Yaskawa INFORM job: OK_R2_O34-37(210,0_180)2AWOK.JBI

/JOB
//NAME OK_R2_O34-37(210,0_180)2AWOK
///FOLDERNAME X4
//POS
///NPOS 226,226,226,7,0,0
///TOOL 0
///POSTYPE PULSE
///PULSE
C00000=-125700,-80476,-34247,159249,27287,28453
C00001=-123130,-74105,-30702,162391,25597,27223
C00002=-122202,-71536,-29217,163608,24992,26738
C00003=-121293,-68396,-25015,165796,25706,25775
C00004=-119897,-67278,-25144,167731,24799,24999
C00005=-121293,-68396,-25015,165796,25706,25775
C00006=-122202,-71536,-29217,163608,24992,26738
C00007=-123284,-67899,-27862,160952,24298,27913
C00008=-122447,-67212,-26586,162727,24486,27140
C00009=-123284,-67899,-27862,160952,24298,27913
C00010=-122202,-71536,-29217,163608,24992,26738
C00011=-123130,-74105,-30702,162391,25597,27223
C00012=-125700,-80476,-34247,159249,27287,28453
C00013=-125517,-80437,-34211,159525,27238,28339
C00014=-122961,-74061,-30663,162666,25556,27108
C00015=-122038,-71489,-29176,163883,24954,26623
C00016=-117667,-71002,-28856,171434,24065,23454
C00017=-117704,-70431,-28835,171227,23800,23550
C00018=-117667,-71002,-28856,171434,24065,23454
C00019=-122038,-71489,-29176,163883,24954,26623
C00020=-119799,-70680,-31927,166276,22459,25716
C00021=-118976,-69928,-30572,168119,22724,24911
C00022=-119799,-70680,-31927,166276,22459,25716
C00023=-122038,-71489,-29176,163883,24954,26623
C00024=-122961,-74061,-30663,162666,25556,27108
C00025=-125517,-80437,-34211,159525,27238,28339
C00026=-140387,-129911,-44763,153839,48320,28262
C00027=-154667,-139794,-63765,132481,63225,34326
C00028=-155865,-52236,-95522,47063,99015,61474
C00029=-122410,-67393,-33433,34982,73766,64939
C00030=-118917,-73983,-33918,35626,69830,65070
C00031=-118508,-70070,-27252,36089,67956,64591
C00032=-117264,-69435,-26201,36204,67200,64847
C00033=-118508,-70070,-27252,36089,67956,64591
C00034=-118437,-72039,-27377,36310,67165,64343
C00035=-118508,-70070,-27252,36089,67956,64591
C00036=-123060,-73487,-31863,35667,70648,63634
C00037=-125159,-74654,-36532,35162,73351,63677
C00038=-117818,-78878,-43515,44751,78217,64927
C00039=-114758,-78477,-39683,45348,75169,64953
C00040=-113298,-77876,-37428,45678,73684,64940
C00041=-114862,-79533,-39394,45465,74705,64688
C00042=-113645,-77017,-38294,45463,74548,65185
C00043=-113477,-77789,-37161,45383,73476,65293
C00044=-119505,-70896,-29485,43711,74626,65290
C00045=-120144,-69706,-28375,43648,74873,65114
C00046=-125052,-63057,-20955,43194,76309,63552
C00047=-128321,-58110,-15632,44166,78560,60322
C00048=-131102,-53426,-10460,43738,79284,59417
C00049=-129277,-58077,-17153,43886,79704,60402
C00050=-131618,-58273,-21031,43272,82484,60567
C00051=-155865,-52236,-95522,47063,99015,61474
C00052=-107841,-78990,-100274,15174,85565,25314
C00053=-120644,-33075,-33747,-17198,86743,-72858
C00054=-120645,-33066,-33740,-17198,86743,-72858
C00055=-121261,-33537,-33634,-17157,86319,-73016
C00056=-120651,-31294,-33185,-17194,87287,-72936
C00057=-120265,-34286,-35568,-17221,87300,-72802
C00058=-121246,-33499,-33406,-17160,86207,-72996
C00059=-120695,-32982,-32791,-17199,86212,-72803
C00060=-123405,-31941,-32460,-10145,86277,-73561
C00061=-120644,-33063,-33738,-17198,86744,-72858
C00062=-120644,-33063,-33738,-17198,86744,-72858
C00063=-120644,-33085,-33753,-9248,85868,-74516
C00064=-120658,-33883,-52020,3249,107968,-57945
C00065=-120634,-51653,-31257,6589,89487,-53974
C00066=-120887,-59194,-41100,6571,91677,-53945
C00067=-114365,-59297,-40540,7297,90721,-51781
C00068=-121686,-52648,-32529,6467,89842,-54312
C00069=-120641,-50150,-31062,6590,90137,-53943
C00070=-115090,-58916,-39821,7220,90542,-52038
C00071=-121020,-51343,-30297,6544,89092,-54127
C00072=-121570,-70600,-40611,7004,74168,-55148
C00073=-127404,-59840,-28957,5949,73181,-57087
C00074=-128623,-57920,-26766,5993,72907,-57518
C00075=-120636,-51546,-31197,-12806,84757,-45971
C00076=-120635,-51562,-31206,-12806,84754,-45970
C00077=-120637,-51473,-31156,-31547,98354,-39015
C00078=-120638,-51464,-31151,-31547,98355,-39016
C00079=-127651,-66621,-42293,-29165,87585,-39205
C00080=-120645,-49986,-30969,-31614,98908,-39175
C00081=-120184,-52981,-33063,-31488,98864,-38978
C00082=-126387,-66657,-42132,-29030,87918,-38805
C00083=-124162,-65853,-41061,-28777,88461,-38095
C00084=-123779,-65431,-40746,-28731,88612,-37988
C00085=-116886,-63013,-38039,-27795,90542,-35857
C00086=-116876,-68393,-50736,-27992,95034,-36929
C00087=-127335,-91521,-66356,2133,76505,-53999
C00088=-120632,-51605,-31230,12938,89151,-58072
C00089=-122382,-77541,-49676,15704,77889,-41459
C00090=-116417,-82504,-50333,15734,74684,-39769
C00091=-121684,-52600,-32501,12821,89583,-58390
C00092=-120640,-50101,-31034,12940,89789,-58008
C00093=-117566,-82113,-49782,15768,74770,-40162
C00094=-137736,-66681,-32025,26351,79133,-47852
C00095=-137780,-65826,-31188,26317,79067,-47879
C00096=-127334,-50999,-24101,13599,84251,-46609
C00097=-127274,-55905,-35607,13545,88687,-46195
C00098=-120633,-51614,-31235,12938,89150,-58073
C00099=-120634,-51391,-31110,-31547,98367,-39018
C00100=-120635,-51381,-31104,-31548,98368,-39018
C00101=-123679,-52106,-31631,-32185,97183,-39896
C00102=-120642,-49903,-30922,-31614,98921,-39177
C00103=-120181,-52898,-33017,-31489,98878,-38981
C00104=-120835,-59376,-36016,-31166,93226,-37672
C00105=-121613,-72530,-44193,-30286,84455,-35757
C00106=-118747,-61104,-37303,-26246,91458,-36794
C00107=-120635,-51379,-31103,-26471,93957,-42710
C00108=-120633,-51391,-31110,-26470,93955,-42709
C00109=-120630,-51586,-31219,10910,92232,-53915
C00110=-120632,-51644,-31252,6564,89533,-53910
C00111=-103812,-53067,-78891,-39071,105659,-38988
C00112=-91163,-136711,-112609,-36408,93269,-29237
C00113=-91163,-136711,-112609,-36408,93269,-29237
C00114=-91163,-136711,-112609,-36408,93269,-29237
C00115=-91163,-136711,-112609,-36408,93269,-29237
C00116=-14735,-147183,-53705,-96059,99176,-32960
C00117=-116063,-75069,-24786,-161373,30180,-27192
C00118=-118646,-74586,-30917,-162370,25797,-27057
C00119=-119577,-72016,-29437,-163583,25187,-26574
C00120=-122851,-69134,-26289,-169408,24955,-24114
C00121=-122803,-67500,-26251,-168862,24172,-24377
C00122=-122851,-69134,-26289,-169408,24955,-24114
C00123=-119577,-72016,-29437,-163583,25187,-26574
C00124=-119782,-71043,-35943,-152224,16280,-31420
C00125=-121147,-70052,-34044,-156561,16387,-29537
C00126=-119067,-67658,-29205,-160988,23362,-27785
C00127=-119577,-72016,-29437,-163583,25187,-26574
C00128=-118646,-74586,-30917,-162370,25797,-27057
C00129=-116063,-80958,-34447,-159238,27499,-28281
C00130=-116167,-79884,-33984,-159178,27227,-28326
C00131=-118709,-73507,-30415,-162283,25553,-27108
C00132=-119627,-70935,-28920,-163488,24953,-26627
C00133=-124970,-68554,-27226,-172714,23781,-22752
C00134=-124929,-67933,-27226,-172492,23472,-22855
C00135=-124970,-68554,-27226,-172714,23781,-22752
C00136=-119627,-70935,-28920,-163488,24953,-26627
C00137=-114841,-73408,-48022,-82057,16864,-69970
C00138=-115635,-73012,-47011,-83260,16231,-69454
C00139=-119724,-68827,-29398,-162557,23640,-27094
C00140=-119627,-70935,-28920,-163488,24953,-26627
C00141=-118709,-73507,-30415,-162283,25553,-27108
C00142=-116167,-79884,-33984,-159178,27227,-28326
C00143=-99237,-131925,-44709,-152289,49940,-28409
C00144=-62709,-186403,-96766,-116405,74373,-39052
C00145=-70314,-132957,-105748,-65746,79738,-62154
C00146=-61806,-120643,-118554,-32165,89559,-74963
C00147=-100254,-58589,-20850,-47462,84028,-58675
C00148=-101968,-51866,-3168,-48574,78104,-56512
C00149=-101968,-51553,-2632,-48598,77990,-56453
C00150=-101518,-52976,-2809,-48578,77787,-56140
C00151=-101968,-51553,-2632,-48598,77990,-56453
C00152=-103386,-50149,-432,-49034,76876,-56530
C00153=-101968,-51553,-2632,-48598,77990,-56453
C00154=-100254,-58589,-20850,-47462,84028,-58675
C00155=-120623,-69117,-28104,-48531,104993,-26022
C00156=-124022,-87503,-41913,-47197,93373,-21899
C00157=-120632,-67990,-28310,-48704,105465,-26277
C00158=-119274,-70289,-29410,-48044,105816,-25785
C00159=-123549,-87206,-41537,-47050,93555,-21770
C00160=-115351,-77678,-31893,-44276,96770,-19561
C00161=-115180,-76774,-30982,-44204,96783,-19491
C00162=-107611,-66250,-20317,-41245,99360,-17323
C00163=-104022,-60066,-14079,-39703,100393,-16240
C00164=-107611,-77742,-40705,-42371,104385,-19399
C00165=-61806,-120643,-118554,-32165,89559,-74963
C00166=-96268,-101177,-113144,-8865,97124,-11070
C00167=-120641,-42853,-51550,17560,92173,73840
C00168=-120646,-33870,-34272,17525,86425,73017
C00169=-119942,-58321,-47290,17224,67969,70679
C00170=-121031,-35101,-36097,17549,86977,72960
C00171=-120651,-32098,-33726,17520,86975,73094
C00172=-121087,-58091,-46777,17546,68025,70253
C00173=-122899,-57278,-45773,18035,68227,69595
C00174=-123358,-56945,-45288,18164,68208,69418
C00175=-121878,-55895,-44787,12232,67936,69995
C00176=-118961,-54720,-57543,10936,75808,71809
C00177=-120654,-86347,-59671,-2864,63718,59361
C00178=-125912,-56068,-36753,-6250,87624,52842
C00179=-128066,-58011,-42816,-6649,92655,51740
C00180=-129226,-58813,-41203,-6752,91180,51406
C00181=-120642,-50370,-31189,-6165,90024,54116
C00182=-119584,-52858,-32650,-6041,89726,54489
C00183=-128796,-58655,-40767,-6707,91029,51560
C00184=-122766,-51369,-31065,-6034,89291,53691
C00185=-122762,-63238,-38041,-5894,80464,54098
C00186=-119550,-58975,-32943,-5845,79752,55225
C00187=-122768,-60053,-29242,1998,72011,53401
C00188=-124703,-66651,-43936,2040,77707,52830
C00189=-120638,-51944,-31419,32003,97998,39113
C00190=-120639,-51928,-31410,32003,98001,39113
C00191=-118996,-52516,-31682,32334,97265,39558
C00192=-121098,-53452,-33319,31944,98508,39075
C00193=-120645,-50452,-31236,32066,98559,39271
C00194=-119173,-52749,-31833,32295,97308,39501
C00195=-119801,-52482,-32070,32192,97780,39386
C00196=-119899,-52107,-31634,32164,97752,39338
C00197=-119950,-60824,-38736,26131,92333,38222
C00198=-119950,-65442,-50997,26401,96995,39269
C00199=-116899,-68263,-56336,11454,97179,48279
C00200=-127404,-81706,-52066,-14147,73081,57801
C00201=-116720,-79858,-46664,-24697,73771,62487
C00202=-120640,-50459,-31240,-12516,89696,58190
C00203=-119581,-52948,-32700,-12396,89486,58575
C00204=-115512,-79082,-45759,-25163,74038,62927
C00205=-108001,-68814,-34854,-26331,75228,65611
C00206=-108064,-68383,-34491,-26332,75206,65593
C00207=-103624,-60475,-25996,-26279,75513,67180
C00208=-112718,-64474,-31424,-18064,72408,63442
C00209=-112718,-70905,-44852,-17685,77140,62731
C00210=-112718,-71186,-45475,-17671,77368,62698
C00211=-120385,-74764,-48938,3443,103646,-6733
C00212=-120303,-75998,-49738,3392,102861,-6716
C00213=-118985,-76178,-48936,3795,102220,-6275
C00214=-121095,-53483,-33336,3688,117233,-6601
C00215=-120643,-50483,-31254,3935,117471,-6417
C00216=-122593,-74979,-47472,2658,102081,-7526
C00217=-122814,-74696,-47089,2584,101998,-7604
C00218=-129478,-71737,-44300,477,101932,-9900
C00219=-129478,-75128,-51887,483,104859,-9888
C00220=-120632,-52031,-31468,10348,93078,-4644
C00221=-120631,-51970,-31434,-12514,89052,58257
C00222=-126964,-95845,-81485,3515,87950,51222
C00223=-130419,-125155,-112371,3575,92040,50165
C00224=-16344,-125828,-114775,3579,93173,50196
C00225=-16344,-125828,-114775,3579,93173,50196
BC00000=299799,668083,634815
BC00001=299799,668083,634815
BC00002=299799,668083,634815
BC00003=299799,668083,634815
BC00004=299799,668083,634815
BC00005=299799,668083,634815
BC00006=299799,668083,634815
BC00007=299799,668083,634815
BC00008=299799,668083,634815
BC00009=299799,668083,634815
BC00010=299799,668083,634815
BC00011=299799,668083,634815
BC00012=299799,668083,634815
BC00013=258861,679019,566863
BC00014=258861,679019,566863
BC00015=258861,679019,566863
BC00016=258861,679019,566863
BC00017=258861,679019,566863
BC00018=258861,679019,566863
BC00019=258861,679019,566863
BC00020=258861,679019,566863
BC00021=258861,679019,566863
BC00022=258861,679019,566863
BC00023=258861,679019,566863
BC00024=258861,679019,566863
BC00025=258861,679019,566863
BC00026=258861,679019,566863
BC00027=246190,684484,603571
BC00028=168329,718064,829131
BC00029=168329,806325,829131
BC00030=168329,806325,829131
BC00031=168329,806325,829131
BC00032=168329,806325,829131
BC00033=168329,806325,829131
BC00034=168329,806325,829131
BC00035=168329,806325,829131
BC00036=168329,806325,829131
BC00037=168329,806325,829131
BC00038=161625,808865,790208
BC00039=161625,808865,790208
BC00040=161625,808865,790208
BC00041=161625,808865,790208
BC00042=161625,808865,790208
BC00043=161625,808865,790208
BC00044=161625,808865,790208
BC00045=161625,808865,790208
BC00046=161625,808865,790208
BC00047=161625,808865,790208
BC00048=161625,808865,790208
BC00049=161625,808865,790208
BC00050=161625,808865,790208
BC00051=168329,718064,829131
BC00052=233669,718722,855431
BC00053=356753,719962,904973
BC00054=355561,717940,879352
BC00055=355084,717131,869103
BC00056=355084,717131,869103
BC00057=355084,717131,869103
BC00058=358688,717759,865405
BC00059=358688,717759,865405
BC00060=358688,717759,865405
BC00061=360357,720590,901274
BC00062=360145,720879,899518
BC00063=353052,720476,901588
BC00064=275657,749180,834890
BC00065=252725,782753,902871
BC00066=256148,780353,880096
BC00067=257517,779394,870985
BC00068=257517,779394,870985
BC00069=257517,779394,870985
BC00070=257517,779394,870985
BC00071=257517,779394,870985
BC00072=257517,779394,870985
BC00073=257517,779394,870985
BC00074=257517,779394,870985
BC00075=279626,776550,839590
BC00076=278375,777634,865867
BC00077=302522,799758,822544
BC00078=301330,797736,796923
BC00079=300854,796928,786673
BC00080=300853,796927,786675
BC00081=300853,796927,786675
BC00082=300854,796928,786673
BC00083=300854,796928,786673
BC00084=300854,796928,786673
BC00085=300854,796928,786673
BC00086=300854,796928,786673
BC00087=285946,783794,900084
BC00088=276545,775017,942522
BC00089=280455,772329,921075
BC00090=280455,772329,921075
BC00091=282019,771253,912497
BC00092=282019,771253,912497
BC00093=280455,772329,921075
BC00094=280455,772329,921075
BC00095=280455,772329,921075
BC00096=280455,772329,921075
BC00097=280403,772359,920891
BC00098=268658,779616,914487
BC00099=344074,788201,893588
BC00100=342882,786179,867967
BC00101=342405,785370,857718
BC00102=342405,785370,857718
BC00103=342405,785370,857718
BC00104=342405,785370,857718
BC00105=342405,785370,857718
BC00106=342405,785370,857718
BC00107=345131,781299,876890
BC00108=345652,783183,902892
BC00109=289564,773957,978220
BC00110=261789,777074,937860
BC00111=353536,737917,894599
BC00112=353536,695664,894599
BC00113=353536,695664,894599
BC00114=353536,695664,894599
BC00115=353536,695664,894599
BC00116=166023,670483,663813
BC00117=139859,666970,631611
BC00118=139859,666970,631611
BC00119=139859,666970,631611
BC00120=139859,666970,631611
BC00121=139859,666971,631609
BC00122=139859,666970,631611
BC00123=139859,666970,631611
BC00124=139859,666970,631611
BC00125=139859,666970,631609
BC00126=139859,666970,631611
BC00127=139859,666970,631611
BC00128=139859,666970,631611
BC00129=139859,666970,631611
BC00130=178204,675740,573402
BC00131=178204,675740,573402
BC00132=178204,675740,573402
BC00133=178204,675740,573402
BC00134=178204,675740,573402
BC00135=178204,675740,573402
BC00136=178204,675740,573402
BC00137=178204,675740,573402
BC00138=178204,675740,573402
BC00139=178204,675740,573402
BC00140=178204,675740,573402
BC00141=178204,675740,573402
BC00142=178204,675740,573402
BC00143=178204,675740,573402
BC00144=191883,696660,621052
BC00145=236191,764425,852086
BC00146=260221,801176,958847
BC00147=260221,801176,859111
BC00148=260221,801176,859108
BC00149=260221,801176,859108
BC00150=260221,801176,859108
BC00151=260221,801176,859108
BC00152=260221,801176,859108
BC00153=260221,801176,859108
BC00154=260221,801176,859111
BC00155=271447,845610,763612
BC00156=269989,844590,755462
BC00157=269905,844531,754994
BC00158=269905,844531,754994
BC00159=269989,844590,755462
BC00160=269989,844590,755462
BC00161=269989,844590,755462
BC00162=269989,844590,755462
BC00163=269989,844590,755462
BC00164=269989,844590,755462
BC00165=260221,801176,859111
BC00166=179215,763567,877996
BC00167=81732,718309,900722
BC00168=82982,716309,875111
BC00169=83482,715509,864866
BC00170=83482,715509,864866
BC00171=83482,715509,864866
BC00172=83482,715509,864866
BC00173=83482,715509,864866
BC00174=83482,715509,864866
BC00175=83482,715509,864866
BC00176=83482,715509,864866
BC00177=162723,767201,899794
BC00178=183133,779963,900503
BC00179=180774,777935,868378
BC00180=180772,777936,868380
BC00181=180651,777993,868574
BC00182=180651,777993,868574
BC00183=180772,777936,868380
BC00184=180772,777936,868380
BC00185=180772,777936,868380
BC00186=180772,777936,868380
BC00187=180772,777936,868380
BC00188=180772,777936,868380
BC00189=135124,798065,819777
BC00190=136374,796066,794166
BC00191=136671,795591,788088
BC00192=136874,795266,783921
BC00193=136874,795266,783921
BC00194=136199,795636,787117
BC00195=132017,796135,779854
BC00196=132017,796135,779854
BC00197=132017,796135,779854
BC00198=132017,796135,779854
BC00199=143790,787140,843333
BC00200=157760,770823,917898
BC00201=157760,770823,917898
BC00202=156218,769744,909280
BC00203=156218,769744,909280
BC00204=157760,770823,917898
BC00205=157760,770824,917897
BC00206=157760,770824,917897
BC00207=157760,770824,917897
BC00208=157760,770824,917897
BC00209=157760,770824,917897
BC00210=157760,770824,917897
BC00211=135405,814938,885725
BC00212=136655,812939,860113
BC00213=136655,812939,860113
BC00214=137155,812139,849869
BC00215=137155,812139,849869
BC00216=136655,812939,860113
BC00217=136655,812939,860113
BC00218=136655,812939,860113
BC00219=136655,812939,860113
BC00220=125409,766237,942300
BC00221=152567,767692,974231
BC00222=182902,779158,882705
BC00223=182902,779158,882705
BC00224=182902,779158,882705
BC00225=182902,668970,882705
EC00000=1862365,0
EC00001=1862365,0
EC00002=1862365,0
EC00003=1862365,0
EC00004=1862365,0
EC00005=1862365,0
EC00006=1862365,0
EC00007=1862365,0
EC00008=1862365,0
EC00009=1862365,0
EC00010=1862365,0
EC00011=1862365,0
EC00012=1862365,0
EC00013=1862365,0
EC00014=1862365,0
EC00015=1862365,0
EC00016=1862365,0
EC00017=1862365,0
EC00018=1862365,0
EC00019=1862365,0
EC00020=1862365,0
EC00021=1862365,0
EC00022=1862365,0
EC00023=1862365,0
EC00024=1862365,0
EC00025=1862365,0
EC00026=1862365,0
EC00027=1862365,0
EC00028=1862365,0
EC00029=1862365,0
EC00030=1862365,0
EC00031=1862365,0
EC00032=1862365,0
EC00033=1862365,0
EC00034=1862365,0
EC00035=1862365,0
EC00036=1862365,0
EC00037=1862365,0
EC00038=1862365,0
EC00039=1862365,0
EC00040=1862365,0
EC00041=1862365,0
EC00042=1862365,0
EC00043=1862365,0
EC00044=1862365,0
EC00045=1862365,0
EC00046=1862365,0
EC00047=1862365,0
EC00048=1862365,0
EC00049=1862365,0
EC00050=1862365,0
EC00051=1862365,0
EC00052=1862365,0
EC00053=1862365,0
EC00054=1862365,0
EC00055=1862365,0
EC00056=1862365,0
EC00057=1862365,0
EC00058=1862365,0
EC00059=1862365,0
EC00060=1862365,0
EC00061=1862365,0
EC00062=1862365,0
EC00063=1862365,0
EC00064=1862365,0
EC00065=1862365,0
EC00066=1862365,0
EC00067=1862365,0
EC00068=1862365,0
EC00069=1862365,0
EC00070=1862365,0
EC00071=1862365,0
EC00072=1862365,0
EC00073=1862365,0
EC00074=1862365,0
EC00075=1862365,0
EC00076=1862365,0
EC00077=1862365,0
EC00078=1862365,0
EC00079=1862365,0
EC00080=1862365,0
EC00081=1862365,0
EC00082=1862365,0
EC00083=1862365,0
EC00084=1862365,0
EC00085=1862365,0
EC00086=1862365,0
EC00087=1862365,0
EC00088=1862365,0
EC00089=1862365,0
EC00090=1862365,0
EC00091=1862365,0
EC00092=1862365,0
EC00093=1862365,0
EC00094=1862365,0
EC00095=1862365,0
EC00096=1862365,0
EC00097=1862365,0
EC00098=1862365,0
EC00099=1862365,0
EC00100=1862365,0
EC00101=1862365,0
EC00102=1862365,0
EC00103=1862365,0
EC00104=1862365,0
EC00105=1862365,0
EC00106=1862365,0
EC00107=1862365,0
EC00108=1862365,0
EC00109=1862365,0
EC00110=1862365,0
EC00111=1862365,0
EC00112=1862365,0
EC00113=1596313,0
EC00114=1596313,1112951
EC00115=1862365,1112951
EC00116=1862365,1112951
EC00117=1862365,1112951
EC00118=1862365,1112951
EC00119=1862365,1112951
EC00120=1862365,1112951
EC00121=1862365,1112952
EC00122=1862365,1112951
EC00123=1862365,1112951
EC00124=1862365,1112951
EC00125=1862366,1112951
EC00126=1862365,1112951
EC00127=1862365,1112951
EC00128=1862365,1112951
EC00129=1862365,1112951
EC00130=1862365,1112951
EC00131=1862365,1112951
EC00132=1862365,1112951
EC00133=1862365,1112951
EC00134=1862365,1112951
EC00135=1862365,1112951
EC00136=1862365,1112951
EC00137=1862365,1112951
EC00138=1862365,1112951
EC00139=1862365,1112951
EC00140=1862365,1112951
EC00141=1862365,1112951
EC00142=1862365,1112951
EC00143=1862365,1112951
EC00144=1862365,1112951
EC00145=1862365,1112951
EC00146=1862365,1112951
EC00147=1862366,1112951
EC00148=1862367,1112952
EC00149=1862367,1112952
EC00150=1862367,1112952
EC00151=1862367,1112952
EC00152=1862367,1112952
EC00153=1862367,1112952
EC00154=1862366,1112951
EC00155=1862365,1112951
EC00156=1862365,1112951
EC00157=1862365,1112951
EC00158=1862365,1112951
EC00159=1862365,1112951
EC00160=1862365,1112951
EC00161=1862365,1112951
EC00162=1862365,1112951
EC00163=1862365,1112951
EC00164=1862365,1112951
EC00165=1862365,1112951
EC00166=1862365,1112951
EC00167=1862365,1112951
EC00168=1862365,1112951
EC00169=1862365,1112951
EC00170=1862365,1112951
EC00171=1862365,1112951
EC00172=1862365,1112951
EC00173=1862365,1112951
EC00174=1862365,1112951
EC00175=1862365,1112951
EC00176=1862365,1112951
EC00177=1862365,1112951
EC00178=1862365,1112951
EC00179=1862365,1112951
EC00180=1862367,1112951
EC00181=1862365,1112951
EC00182=1862365,1112951
EC00183=1862367,1112951
EC00184=1862367,1112951
EC00185=1862367,1112951
EC00186=1862367,1112951
EC00187=1862367,1112951
EC00188=1862367,1112951
EC00189=1862365,1112951
EC00190=1862365,1112951
EC00191=1862365,1112951
EC00192=1862365,1112951
EC00193=1862365,1112951
EC00194=1862365,1112951
EC00195=1862365,1112951
EC00196=1862365,1112951
EC00197=1862365,1112951
EC00198=1862365,1112951
EC00199=1862365,1112951
EC00200=1862365,1112951
EC00201=1862365,1112951
EC00202=1862365,1112951
EC00203=1862365,1112951
EC00204=1862365,1112951
EC00205=1862367,1112951
EC00206=1862367,1112951
EC00207=1862367,1112951
EC00208=1862367,1112951
EC00209=1862367,1112951
EC00210=1862367,1112951
EC00211=1862365,1112951
EC00212=1862365,1112951
EC00213=1862365,1112951
EC00214=1862365,1112951
EC00215=1862365,1112951
EC00216=1862365,1112951
EC00217=1862365,1112951
EC00218=1862365,1112951
EC00219=1862365,1112951
EC00220=1862365,1112951
EC00221=1862365,1112951
EC00222=1862365,1112951
EC00223=1862365,1112951
EC00224=1862365,1112951
EC00225=1862365,1112951
///POSTYPE BASE
///RECTAN
///RCONF 0,0,0,0,0,0,0,0,0,0,0,0,0,0,0,0,0,0,0,0,0,0,0,0
P00006=0.222,-3.123,-1.508,0.0000,0.0000,0.0000
P00021=-0.225,-6.128,-0.405,0.0000,0.0000,0.0000
P00022=0.222,-3.123,-1.508,0.0000,0.0000,0.0000
P00023=0.143,-0.036,0.682,0.0000,0.0000,0.0000
P00031=1.853,-0.001,-1.549,0.0000,0.0000,0.0000
P00032=1.957,0.503,-7.217,0.0000,0.0000,0.0000
///RCONF 0,0,0,0,1,0,0,0,0,0,0,0,0,0,0,0,0,0,0,0,0,0,0,0
P00033=-0.123,0.612,-5.012,0.0000,0.0000,0.0000
//INST
///DATE 2024/02/13 20:40
///ATTR SC,RW
///GROUP1 RB1,BS1
///GROUP2 ST1
NOP
'OK_r2_O34-37(-90,0_180)2
'210,0
'Path S1900
SFTOF3D
MOVJ C00000 BC00000 VJ=100.00  +MOVJ EC00000 VJ=100.00
MOVL C00001 BC00001 V=400.0  +MOVJ EC00001 VJ=100.00
SMOVL C00002 BC00002 V=100.0  +MOVJ EC00002
SMOVL C00003 BC00003 V=60.0  +MOVJ EC00003
SREFP 3 C00004 BC00004  +REFP EC00004
CALL JOB:SEARCH-R1-S13D
SET P023 P006
SFTON3D P023
SMOVL C00005 BC00005 V=60.0  +MOVJ EC00005
SMOVL C00006 BC00006 V=100.0  +MOVJ EC00006
SMOVL C00007 BC00007 V=60.0  +MOVJ EC00007
SREFP 3 C00008 BC00008  +REFP EC00008
CALL JOB:SEARCH-R1-S13D
SET P023 P006
SFTON3D P023
SMOVL C00009 BC00009 V=60.0  +MOVJ EC00009
SMOVL C00010 BC00010 V=100.0  +MOVJ EC00010
MOVL C00011 BC00011 V=400.0  +MOVJ EC00011 VJ=100.00
MOVL C00012 BC00012 V=1000.0  +MOVJ EC00012 VJ=100.00
'Path S1899
SFTOF3D
MOVJ C00013 BC00013 VJ=100.00  +MOVJ EC00013 VJ=100.00
MOVL C00014 BC00014 V=400.0  +MOVJ EC00014 VJ=100.00
SMOVL C00015 BC00015 V=100.0  +MOVJ EC00015
SMOVL C00016 BC00016 V=60.0  +MOVJ EC00016
SREFP 3 C00017 BC00017  +REFP EC00017
CALL JOB:SEARCH-R1-S13D
SET P022 P006
SFTON3D P022
SMOVL C00018 BC00018 V=60.0  +MOVJ EC00018
SMOVL C00019 BC00019 V=100.0  +MOVJ EC00019
SMOVL C00020 BC00020 V=60.0  +MOVJ EC00020
SREFP 3 C00021 BC00021  +REFP EC00021
CALL JOB:SEARCH-R1-S13D
SET P022 P006
SFTON3D P022
SMOVL C00022 BC00022 V=60.0  +MOVJ EC00022
SMOVL C00023 BC00023 V=100.0  +MOVJ EC00023
MOVL C00024 BC00024 V=400.0  +MOVJ EC00024 VJ=100.00
MOVL C00025 BC00025 V=1000.0  +MOVJ EC00025 VJ=100.00
MOVJ C00026 BC00026 VJ=100.00  +MOVJ EC00026 VJ=100.00
MOVJ C00027 BC00027 VJ=100.00  +MOVJ EC00027 VJ=100.00
MOVJ C00028 BC00028 VJ=100.00  +MOVJ EC00028 VJ=100.00
'Path S1903
SFTOF3D
MOVJ C00029 BC00029 VJ=100.00  +MOVJ EC00029 VJ=100.00
MOVL C00030 BC00030 V=400.0  +MOVJ EC00030 VJ=100.00
SMOVL C00031 BC00031 V=60.0  +MOVJ EC00031
SREFP 3 C00032 BC00032  +REFP EC00032
CALL JOB:SEARCH-R1-S13D
SET P021 P006
SFTON3D P021
SMOVL C00033 BC00033 V=60.0  +MOVJ EC00033
SREFP 3 C00034 BC00034  +REFP EC00034
CALL JOB:SEARCH-R1-S13D
SET P021 P006
SFTON3D P021
SMOVL C00035 BC00035 V=60.0  +MOVJ EC00035
MOVL C00036 BC00036 V=400.0  +MOVJ EC00036 VJ=100.00
MOVL C00037 BC00037 V=1000.0  +MOVJ EC00037 VJ=100.00
'Path W1908
SFTOF3D
PAUSE
SFTON3D P021
MOVJ C00038 BC00038 VJ=100.00  +MOVJ EC00038 VJ=100.00
SMOVL C00039 BC00039 V=100.0  +MOVJ EC00039
SMOVL C00040 BC00040 V=100.0 PL=0  +MOVJ EC00040
SREFP 1 C00041 BC00041  +REFP EC00041
SREFP 2 C00042 BC00042  +REFP EC00042
MACRO1 MJ#(0) ARGF14
ARCON
SMOVL C00043 BC00043 V=11.7  +MOVJ EC00043
SMOVL C00044 BC00044 V=11.7  +MOVJ EC00044
SMOVL C00045 BC00045 V=11.7  +MOVJ EC00045
SMOVL C00046 BC00046 V=11.7  +MOVJ EC00046
SMOVL C00047 BC00047 V=11.7  +MOVJ EC00047
ARCON
SMOVL C00048 BC00048 V=11.7  +MOVJ EC00048
ARCOF
SMOVL C00049 BC00049 V=400.0  +MOVJ EC00049
SMOVL C00050 BC00050 V=1000.0  +MOVJ EC00050
SFTOF3D
MOVJ C00051 BC00051 VJ=40.00  +MOVJ EC00051 VJ=100.00
MOVJ C00052 BC00052 VJ=100.00  +MOVJ EC00052 VJ=100.00
'Path W1909
SFTOF3D
SFTON3D P023
MOVJ C00053 BC00053 VJ=100.00  +MOVJ EC00053 VJ=100.00
SMOVL C00054 BC00054 V=100.0  +MOVJ EC00054
SMOVL C00055 BC00055 V=100.0 PL=0  +MOVJ EC00055
SREFP 1 C00056 BC00056  +REFP EC00056
SREFP 2 C00057 BC00057  +REFP EC00057
MACRO1 MJ#(0) ARGF6
ARCON
SMOVL C00058 BC00058 V=10.0  +MOVJ EC00058
SMOVL C00059 BC00059 V=10.0  +MOVJ EC00059
SMOVL C00060 BC00060 V=10.0  +MOVJ EC00060
ARCOF
SMOVL C00061 BC00061 V=166.7  +MOVJ EC00061
SFTOF3D
'Path W1910
SFTOF3D
SFTON3D P023
MOVJ C00062 BC00062 VJ=100.00  +MOVJ EC00062 VJ=100.00
SMOVL C00063 BC00063 V=1000.0  +MOVJ EC00063
SFTOF3D
MOVJ C00064 BC00064 VJ=100.00  +MOVJ EC00064 VJ=100.00
'Path W1911
SFTOF3D
SFTON3D P022
MOVJ C00065 BC00065 VJ=100.00  +MOVJ EC00065 VJ=100.00
SMOVL C00066 BC00066 V=100.0  +MOVJ EC00066
SMOVL C00067 BC00067 V=100.0 PL=0  +MOVJ EC00067
SREFP 1 C00068 BC00068  +REFP EC00068
SREFP 2 C00069 BC00069  +REFP EC00069
MACRO1 MJ#(0) ARGF6
ARCON
SMOVL C00070 BC00070 V=10.0  +MOVJ EC00070
SMOVL C00071 BC00071 V=10.0  +MOVJ EC00071
SMOVL C00072 BC00072 V=10.0  +MOVJ EC00072
SMOVL C00073 BC00073 V=10.0  +MOVJ EC00073
SMOVL C00074 BC00074 V=10.0  +MOVJ EC00074
ARCOF
SMOVL C00075 BC00075 V=400.0  +MOVJ EC00075
SMOVL C00076 BC00076 V=1000.0  +MOVJ EC00076
SFTOF3D
'Path W1912
SFTOF3D
SFTON3D P021
MOVJ C00077 BC00077 VJ=100.00  +MOVJ EC00077 VJ=100.00
SMOVL C00078 BC00078 V=100.0  +MOVJ EC00078
SMOVL C00079 BC00079 V=100.0 PL=0  +MOVJ EC00079
SREFP 1 C00080 BC00080  +REFP EC00080
SREFP 2 C00081 BC00081  +REFP EC00081
MACRO1 MJ#(0) ARGF6
ARCON
SMOVL C00082 BC00082 V=10.0  +MOVJ EC00082
SMOVL C00083 BC00083 V=10.0  +MOVJ EC00083
SMOVL C00084 BC00084 V=10.0  +MOVJ EC00084
SMOVL C00085 BC00085 V=10.0  +MOVJ EC00085
ARCOF
SMOVL C00086 BC00086 V=400.0  +MOVJ EC00086
SFTOF3D
'Path W1913
MOVJ C00087 BC00087 VJ=100.00  +MOVJ EC00087 VJ=100.00
'Path W1914
SFTOF3D
SFTON3D P023
MOVJ C00088 BC00088 VJ=100.00  +MOVJ EC00088 VJ=100.00
SMOVL C00089 BC00089 V=100.0  +MOVJ EC00089
SMOVL C00090 BC00090 V=100.0 PL=0  +MOVJ EC00090
SREFP 1 C00091 BC00091  +REFP EC00091
SREFP 2 C00092 BC00092  +REFP EC00092
MACRO1 MJ#(0) ARGF6
ARCON
SMOVL C00093 BC00093 V=10.0  +MOVJ EC00093
SMOVL C00094 BC00094 V=10.0  +MOVJ EC00094
SMOVL C00095 BC00095 V=10.0  +MOVJ EC00095
SMOVL C00096 BC00096 V=10.0  +MOVJ EC00096
ARCOF
SMOVL C00097 BC00097 V=400.0  +MOVJ EC00097
SMOVL C00098 BC00098 V=1000.0  +MOVJ EC00098
SFTOF3D
'Path W1915
SFTOF3D
SFTON3D P023
MOVJ C00099 BC00099 VJ=100.00  +MOVJ EC00099 VJ=100.00
SMOVL C00100 BC00100 V=100.0  +MOVJ EC00100
SMOVL C00101 BC00101 V=100.0 PL=0  +MOVJ EC00101
SREFP 1 C00102 BC00102  +REFP EC00102
SREFP 2 C00103 BC00103  +REFP EC00103
MACRO1 MJ#(0) ARGF6
ARCON
SMOVL C00104 BC00104 V=10.0  +MOVJ EC00104
SMOVL C00105 BC00105 V=10.0  +MOVJ EC00105
SMOVL C00106 BC00106 V=10.0  +MOVJ EC00106
ARCOF
SMOVL C00107 BC00107 V=400.0  +MOVJ EC00107
SMOVL C00108 BC00108 V=1000.0  +MOVJ EC00108
SFTOF3D
SFTOF3D
'Path W1901
SFTOF3D
SFTON3D P023
MOVJ C00109 BC00109 VJ=100.00  +MOVJ EC00109 VJ=100.00
SFTOF3D
SFTON3D P022
MOVJ C00110 BC00110 VJ=100.00  +MOVJ EC00110 VJ=100.00
SFTOF3D
SFTON3D P023
SFTOF3D
MOVJ C00111 BC00111 VJ=100.00  +MOVJ EC00111 VJ=100.00
MOVJ C00112 BC00112 VJ=100.00  +MOVJ EC00112 VJ=100.00
MOVJ C00113 BC00113 VJ=100.00  +MOVJ EC00113 VJ=100.00
MOVJ C00114 BC00114 VJ=100.00  +MOVJ EC00114 VJ=100.00
MOVJ C00115 BC00115 VJ=100.00  +MOVJ EC00115 VJ=100.00
CALL JOB:CLEAN-R1_KM
MOVJ C00116 BC00116 VJ=100.00  +MOVJ EC00116 VJ=100.00
'210,180
'Path S1905
SFTOF3D
MOVJ C00117 BC00117 VJ=100.00  +MOVJ EC00117 VJ=100.00
MOVL C00118 BC00118 V=400.0  +MOVJ EC00118 VJ=100.00
SMOVL C00119 BC00119 V=100.0  +MOVJ EC00119
SMOVL C00120 BC00120 V=60.0  +MOVJ EC00120
SREFP 3 C00121 BC00121  +REFP EC00121
CALL JOB:SEARCH-R1-S13D
SET P033 P006
SFTON3D P033
SMOVL C00122 BC00122 V=60.0  +MOVJ EC00122
SMOVL C00123 BC00123 V=100.0  +MOVJ EC00123
SMOVL C00124 BC00124 V=60.0  +MOVJ EC00124
SREFP 3 C00125 BC00125  +REFP EC00125
CALL JOB:SEARCH-R1-S13D
SET P033 P006
SFTON3D P033
SMOVL C00126 BC00126 V=60.0  +MOVJ EC00126
SMOVL C00127 BC00127 V=100.0  +MOVJ EC00127
MOVL C00128 BC00128 V=400.0  +MOVJ EC00128 VJ=100.00
MOVL C00129 BC00129 V=1000.0  +MOVJ EC00129 VJ=100.00
'Path S1904
SFTOF3D
MOVJ C00130 BC00130 VJ=100.00  +MOVJ EC00130 VJ=100.00
MOVL C00131 BC00131 V=400.0  +MOVJ EC00131 VJ=100.00
SMOVL C00132 BC00132 V=100.0  +MOVJ EC00132
SMOVL C00133 BC00133 V=60.0  +MOVJ EC00133
SREFP 3 C00134 BC00134  +REFP EC00134
CALL JOB:SEARCH-R1-S13D
SET P032 P006
SFTON3D P032
SMOVL C00135 BC00135 V=60.0  +MOVJ EC00135
SMOVL C00136 BC00136 V=100.0  +MOVJ EC00136
SMOVL C00137 BC00137 V=60.0  +MOVJ EC00137
SREFP 3 C00138 BC00138  +REFP EC00138
CALL JOB:SEARCH-R1-S13D
SET P032 P006
SFTON3D P032
SMOVL C00139 BC00139 V=60.0  +MOVJ EC00139
SMOVL C00140 BC00140 V=100.0  +MOVJ EC00140
MOVL C00141 BC00141 V=400.0  +MOVJ EC00141 VJ=100.00
MOVL C00142 BC00142 V=1000.0  +MOVJ EC00142 VJ=100.00
MOVJ C00143 BC00143 VJ=100.00  +MOVJ EC00143 VJ=100.00
MOVJ C00144 BC00144 VJ=100.00  +MOVJ EC00144 VJ=100.00
MOVJ C00145 BC00145 VJ=100.00  +MOVJ EC00145 VJ=100.00
MOVJ C00146 BC00146 VJ=100.00  +MOVJ EC00146 VJ=100.00
'Path S1917
SFTOF3D
MOVJ C00147 BC00147 VJ=50.00  +MOVJ EC00147 VJ=50.00
MOVL C00148 BC00148 V=400.0  +MOVJ EC00148 VJ=100.00
SMOVL C00149 BC00149 V=60.0  +MOVJ EC00149
SREFP 3 C00150 BC00150  +REFP EC00150
CALL JOB:SEARCH-R1-S13D
SET P031 P006
SFTON3D P031
SMOVL C00151 BC00151 V=60.0  +MOVJ EC00151
SREFP 3 C00152 BC00152  +REFP EC00152
CALL JOB:SEARCH-R1-S13D
SET P031 P006
SFTON3D P031
SMOVL C00153 BC00153 V=60.0  +MOVJ EC00153
MOVL C00154 BC00154 V=1000.0  +MOVJ EC00154 VJ=100.00
'Path W1918
SFTOF3D
SFTON3D P031
SMOVL C00155 BC00155 V=400.0  +MOVJ EC00155
SMOVL C00156 BC00156 V=100.0 PL=0  +MOVJ EC00156
SREFP 1 C00157 BC00157  +REFP EC00157
SREFP 2 C00158 BC00158  +REFP EC00158
MACRO1 MJ#(0) ARGF6
ARCON
SMOVL C00159 BC00159 V=10.0  +MOVJ EC00159
SMOVL C00160 BC00160 V=10.0  +MOVJ EC00160
SMOVL C00161 BC00161 V=10.0  +MOVJ EC00161
SMOVL C00162 BC00162 V=10.0  +MOVJ EC00162
ARCON
SMOVL C00163 BC00163 V=10.0  +MOVJ EC00163
ARCOF
SMOVL C00164 BC00164 V=400.0  +MOVJ EC00164
SFTOF3D
MOVJ C00165 BC00165 VJ=100.00  +MOVJ EC00165 VJ=100.00
MOVJ C00166 BC00166 VJ=100.00  +MOVJ EC00166 VJ=100.00
'Path W1919
SFTOF3D
SFTON3D P033
MOVJ C00167 BC00167 VJ=100.00  +MOVJ EC00167 VJ=100.00
SMOVL C00168 BC00168 V=400.0  +MOVJ EC00168
SMOVL C00169 BC00169 V=100.0 PL=0  +MOVJ EC00169
SREFP 1 C00170 BC00170  +REFP EC00170
SREFP 2 C00171 BC00171  +REFP EC00171
MACRO1 MJ#(0) ARGF6
ARCON
SMOVL C00172 BC00172 V=10.0  +MOVJ EC00172
SMOVL C00173 BC00173 V=10.0  +MOVJ EC00173
SMOVL C00174 BC00174 V=10.0  +MOVJ EC00174
SMOVL C00175 BC00175 V=10.0  +MOVJ EC00175
ARCOF
SMOVL C00176 BC00176 V=400.0  +MOVJ EC00176
SFTOF3D
MOVJ C00177 BC00177 VJ=100.00  +MOVJ EC00177 VJ=100.00
'Path W1921
SFTOF3D
SFTON3D P032
MOVJ C00178 BC00178 VJ=20.00  +MOVJ EC00178 VJ=100.00
SMOVL C00179 BC00179 V=400.0  +MOVJ EC00179
SMOVL C00180 BC00180 V=100.0 PL=0  +MOVJ EC00180
SREFP 1 C00181 BC00181  +REFP EC00181
SREFP 2 C00182 BC00182  +REFP EC00182
MACRO1 MJ#(0) ARGF6
ARCON
SMOVL C00183 BC00183 V=10.0  +MOVJ EC00183
SMOVL C00184 BC00184 V=10.0  +MOVJ EC00184
SMOVL C00185 BC00185 V=10.0  +MOVJ EC00185
SMOVL C00186 BC00186 V=10.0  +MOVJ EC00186
SMOVL C00187 BC00187 V=10.0  +MOVJ EC00187
ARCOF
SMOVL C00188 BC00188 V=400.0  +MOVJ EC00188
SFTOF3D
'Path W1922
SFTOF3D
SFTON3D P031
MOVJ C00189 BC00189 VJ=100.00  +MOVJ EC00189 VJ=100.00
SMOVL C00190 BC00190 V=400.0  +MOVJ EC00190
SMOVL C00191 BC00191 V=100.0 PL=0  +MOVJ EC00191
SREFP 1 C00192 BC00192  +REFP EC00192
SREFP 2 C00193 BC00193  +REFP EC00193
MACRO1 MJ#(0) ARGF6
ARCON
SMOVL C00194 BC00194 V=10.0  +MOVJ EC00194
SMOVL C00195 BC00195 V=10.0  +MOVJ EC00195
SMOVL C00196 BC00196 V=10.0  +MOVJ EC00196
SMOVL C00197 BC00197 V=10.0  +MOVJ EC00197
ARCOF
SMOVL C00198 BC00198 V=400.0  +MOVJ EC00198
SFTOF3D
SFTON3D P033
MOVJ C00199 BC00199 VJ=100.00  +MOVJ EC00199 VJ=100.00
SMOVL C00200 BC00200 V=400.0  +MOVJ EC00200
SMOVL C00201 BC00201 V=100.0 PL=0  +MOVJ EC00201
SREFP 1 C00202 BC00202  +REFP EC00202
SREFP 2 C00203 BC00203  +REFP EC00203
MACRO1 MJ#(0) ARGF6
ARCON
SMOVL C00204 BC00204 V=10.0  +MOVJ EC00204
SMOVL C00205 BC00205 V=10.0  +MOVJ EC00205
SMOVL C00206 BC00206 V=10.0  +MOVJ EC00206
SMOVL C00207 BC00207 V=10.0  +MOVJ EC00207
SMOVL C00208 BC00208 V=10.0  +MOVJ EC00208
ARCOF
SMOVL C00209 BC00209 V=400.0  +MOVJ EC00209
MOVJ C00210 BC00210 VJ=50.00  +MOVJ EC00210 VJ=50.00
SFTOF3D
'Path W1925
SFTOF3D
SFTON3D P032
MOVJ C00211 BC00211 VJ=100.00  +MOVJ EC00211 VJ=100.00
SMOVL C00212 BC00212 V=400.0  +MOVJ EC00212
SMOVL C00213 BC00213 V=100.0 PL=0  +MOVJ EC00213
SREFP 1 C00214 BC00214  +REFP EC00214
SREFP 2 C00215 BC00215  +REFP EC00215
MACRO1 MJ#(0) ARGF6
ARCON
SMOVL C00216 BC00216 V=10.0  +MOVJ EC00216
SMOVL C00217 BC00217 V=10.0  +MOVJ EC00217
SMOVL C00218 BC00218 V=10.0  +MOVJ EC00218
ARCOF
SMOVL C00219 BC00219 V=400.0  +MOVJ EC00219
SFTOF3D
SFTON3D P032
MOVJ C00220 BC00220 VJ=100.00  +MOVJ EC00220 VJ=100.00
SFTOF3D
SFTON3D P033
MOVJ C00221 BC00221 VJ=100.00  +MOVJ EC00221 VJ=100.00
SFTOF3D
MOVJ C00222 BC00222 VJ=50.00  +MOVJ EC00222 VJ=50.00
MOVJ C00223 BC00223 VJ=50.00  +MOVJ EC00223 VJ=50.00
MOVJ C00224 BC00224 VJ=50.00  +MOVJ EC00224 VJ=50.00
MOVJ C00225 BC00225 VJ=50.00  +MOVJ EC00225 VJ=50.00
END
